Staubli VAL3: delete.pgx

public program delete(string x_sName (dimensions=1), num& x_nResult[] (dimensions=1))
  local num l_nSize
  local string l_sItem
begin
  //
  // delete the select option
  //
  if save:nBoxType==1
    if isDefined(sml:box[x_sName])
      // delete
      delete(sml:box[x_sName])
      // save it
      // bToSave=true
      x_nResult=0
    else
      x_nResult=-1
    endIf
  elseIf save:nBoxType==2
    if isDefined(big:box[x_sName])
      // delete
      delete(big:box[x_sName])
      // save it
      // bToSave=true
      x_nResult=0
    else
      x_nResult=-1
    endIf
  endIf
end
